TYPE ST_ItemPK3_OUT3 :
STRUCT
	Identity		:ST_Identity_PK3_OUT3;
	ItemState		:STRING;
	RejectReason	:ST_RejectReason_PK3_OUT3;
	logs			:ST_logs_PK3_OUT3;
	NoRead			:STRING;
END_STRUCT
END_TYPE

(* stored: Version 1.1.0.1, ProductVersion 3.1.4024.13
   DUT ST_ItemPK3_OUT3: Id {38434f4a-ef19-40e6-8274-0d78d228c7f7} *)
